FUNCTION_BLOCK ConveyorController
VAR_INPUT
	AtBufferEntry : BOOL;
	AtBufferExit : BOOL;
	AtExit : BOOL;
END_VAR
VAR_OUTPUT
	EntryConveyor: BOOL;
	ExitConveyor: BOOL;
END_VAR
VAR
	state: INT;
	TimerTP : TP;
	TimerTOF : TOF;
END_VAR

IF GVL.isSystemON THEN
	CASE state OF
		0: // Box collection stage
			EntryConveyor := TRUE;
			TimerTP(IN := NOT AtBufferExit, PT := T#1200MS, Q => ExitConveyor);
			IF NOT AtExit THEN
				state := 1;
			END_IF;
		1: // Box removal stage
			EntryConveyor := FALSE;
			TimerTOF(IN := NOT AtExit, PT := T#1S, Q => ExitConveyor);
			IF NOT TimerTOF.Q THEN
				state := 0;
			END_IF;
	ELSE
		state := 0;
	END_CASE;
ELSE
	EntryConveyor := FALSE;
	ExitConveyor := FALSE;
	state := 0;
END_IF;

END_FUNCTION_BLOCK

(* stored: Version 1.1.0.1, ProductVersion 3.1.4024.12
   POU ConveyorController: Id {d61dc998-b604-42df-a6c5-73cc5dbd69a1}, SpecialFunc None *)
